(* PLC project Untitled1, Beckhoff Automation GmbH TwinCAT PLC Control 3.5.13.21 *)
(* stored: creationDateTime 2022-05-06T13:52:37.3912797, modificationDateTime 2022-05-06T13:52:37.3942797 *)

PROGRAM AutoImported
  VAR
    Step : INT;
    StepReadEtherCATDiagnostics : INT;
    TonReadDiagnostics : TON;
    sError : STRING;
    FB_EcCoESdoWrite1 : FB_EcCoESdoWrite;
    CoEWriteBuffer : DWORD;
    fbEcGetAllSlaveAbnormalStateChanges : FB_EcGetAllSlaveAbnormalStateChanges;
    fbGetAllSlaveStates : FB_EcGetAllSlaveStates;
    fbEcGetConfSlaves : FB_EcGetConfSlaves;
    fbEcGetAllSlaveCrcErrors : FB_EcGetAllSlaveCrcErrors;
    stSlaveStates : ARRAY[0..dwMaxSlaves] OF ST_EcSlaveState;
    stArrEcConfSlaveInfo : ARRAY[0..dwMaxSlaves] OF ST_EcSlaveConfigData;
    dwArrSlaveCrcCount : ARRAY[0..dwMaxSlaves] OF DWORD;
    dwArrSlaveChangeCount : ARRAY[0..dwMaxSlaves] OF DWORD;
    bExecuteFB_GetAdaptersInfo : BOOL := TRUE;  (* /////// Set IP address////////////// *)
    NICCount : INT := 2;
    NicIndex : INT := 1;
    FB_GetAdaptersInfo : FB_GetAdaptersInfo;
    fbDiagRegister : FB_IPCDiag_Register := (sNetId := '');
    fbWriteNicInfo : FB_IPCDiag_WriteParameter;
    iPrevState : INT;
    iState : INT;
    _usiModuleIndex : USINT;
    _sIPAddress : STRING;
    _sIPSubNetMask : STRING;
    _sIPGateway : STRING;
    _xDHCP : BOOL;
    rtExecuteTrig : R_TRIG;
    xBusy : BOOL;
    xError : BOOL;
    hrErrorCode : HRESULT;
    xExecute : BOOL;
    usiModuleIndex : USINT;
    sIPAddress : STRING;
    sIPSubnetMask : STRING;
    sIPGateway : STRING;
    xDHCP : BOOL;
    sCurrentNicName : STRING;
  END_VAR
  VAR CONSTANT
    dwMaxSlaves : DWORD := 50;
  END_VAR

            EtherCAT_Diagnostics();

SetIpAddress();

CASE Step OF
	0:
		//Not implimented yet.
	
	100:
		IF GVL_AutoGenerated.EtherCAT_CoEWriteExecute THEN
			Step:=Step+10;
		END_IF

		
	110:
	FB_EcCoESdoWrite1(
		sNetId:= , 
		nSlaveAddr:= , 
		nSubIndex:= , 
		nIndex:= , 
		pSrcBuf:= , 
		cbBufLen:= , 
		bExecute:= , 
		tTimeout:= , 
		bBusy=> , 
		bError=> , 
		nErrId=> );
		
	120:
		GVL_AutoGenerated.EtherCAT_CoEWriteDone:=TRUE;
END_CASE


          

METHOD EtherCAT_Diagnostics : BOOL
                  
CASE StepReadEtherCATDiagnostics OF
0:
	fbEcGetAllSlaveAbnormalStateChanges.bExecute:=FALSE;
	fbGetAllSlaveStates.bExecute:=FALSE;
	fbEcGetConfSlaves.bExecute:=FALSE;
	//fbEcGetAllSlaveCrcErrors.bError:=FALSE;
	TonReadDiagnostics(IN:=TRUE, PT:=T#1S);
	IF TonReadDiagnostics.q THEN
		TonReadDiagnostics(IN:=FALSE);
		StepReadEtherCATDiagnostics:=StepReadEtherCATDiagnostics+10;
		fbEcGetAllSlaveAbnormalStateChanges.bExecute:=TRUE;
		fbGetAllSlaveStates.bExecute:=TRUE;
		fbEcGetConfSlaves.bExecute:=TRUE;
		//fbEcGetAllSlaveCrcErrors.bError:=TRUE;
	END_IF

10:
	IF NOT fbEcGetAllSlaveAbnormalStateChanges.bBusy THEN
		StepReadEtherCATDiagnostics:=StepReadEtherCATDiagnostics+10;
		IF NOT fbEcGetAllSlaveAbnormalStateChanges.bError THEN		
			;
		ELSE
			sError:='fbEcGetAllSlaveAbnormalStateChanges';
		END_IF
	END_IF
	
20:
	IF NOT fbGetAllSlaveStates.bBusy THEN
		StepReadEtherCATDiagnostics:=StepReadEtherCATDiagnostics+10;
		IF fbGetAllSlaveStates.bError THEN
			sError:='fbGetAllSlaveStates';
		END_IF
	END_IF
	
30:
	IF NOT fbEcGetConfSlaves.bBusy THEN
		StepReadEtherCATDiagnostics:=StepReadEtherCATDiagnostics+10;
		IF fbEcGetConfSlaves.bError THEN
			sError:='fbEcGetConfSlaves';
		END_IF
	END_IF
	
40:
	IF NOT fbEcGetAllSlaveCrcErrors.bBusy THEN
		StepReadEtherCATDiagnostics:=StepReadEtherCATDiagnostics+10;
		IF fbEcGetAllSlaveCrcErrors.bError THEN			
			sError:='fbEcGetAllSlaveCrcErrors';
		END_IF
	END_IF
	
50:	//Use this step to copy all the values to PDO to be sent to the EIP network
	StepReadEtherCATDiagnostics:=0;
	GVL_AutoGenerated.EtherCATChangeCount[1]:=DWORD_TO_UINT(dwArrSlaveChangeCount[1]);
END_CASE


FB_EcCoESdoWrite1(
	sNetId:= F_CreateAmsNetId(nIds := GVL_AutoGenerated.EtherCAT_NetId) , 
	nSlaveAddr:=GVL_AutoGenerated.EtherCAT_CoEWriteSlaveAddr , 
	nSubIndex:=GVL_AutoGenerated.EtherCAT_CoEWriteSubIndex , 
	nIndex:= GVL_AutoGenerated.EtherCAT_CoEWriteIndex, 
	pSrcBuf:=ADR(CoEWriteBuffer) , 
	cbBufLen:=SIZEOF(CoEWriteBuffer) , 
	bBusy=> , 
	bError=>GVL_AutoGenerated.EtherCAT_CoEWriteError , 
	nErrId=> );

	
fbEcGetAllSlaveAbnormalStateChanges(
	sNetId:= F_CreateAmsNetId(nIds := GVL_AutoGenerated.EtherCAT_NetId), 
	pAddrBuf:= ADR(dwArrSlaveChangeCount), 
	cbBufLen:= SIZEOF(dwArrSlaveChangeCount), 
	bExecute:= , 
	tTimeout:= , 
	bBusy=> , 
	bError=> , 
	nErrId=> , 
	nSlaves=> );

fbGetAllSlaveStates(
	sNetId		:=  F_CreateAmsNetId(nIds := GVL_AutoGenerated.EtherCAT_NetId),
	pStateBuf	:= ADR(stSlaveStates),
	cbBufLen	:= SIZEOF(stSlaveStates),
	//bExecute	:=TRUE ,
	tTimeout	:= T#2s);

fbEcGetConfSlaves(bExecute:=FALSE);
fbEcGetConfSlaves(
	sNetId:=F_CreateAmsNetId(nIds := GVL_AutoGenerated.EtherCAT_NetId),
	pArrEcConfSlaveInfo:=ADR(stArrEcConfSlaveInfo) ,
	cbBufLen:=SIZEOF(stArrEcConfSlaveInfo) ,
	//bExecute:=TRUE ,
	tTimeout:=T#2s  );

fbEcGetAllSlaveCrcErrors(bExecute:=FALSE);
fbEcGetAllSlaveCrcErrors(
	sNetId:=F_CreateAmsNetId(nIds := GVL_AutoGenerated.EtherCAT_NetId) ,
	pCrcErrorBuf:=ADR(dwArrSlaveCrcCount) ,
	cbBufLen:=SIZEOF(dwArrSlaveCrcCount) ,
	//bExecute:=TRUE 
);
	
                
END_METHOD

METHOD SetIpAddress : BOOL
                  rtExecuteTrig(clk:= xExecute);
usiModuleIndex;
//sIPAddress:=GVL_Constants_AutoGenerated.PLCIPAddress;
//sIPSubnetMask:='255.255.255.0';
//xDHCP:=false;
//sIPAddress := PLCIPAddress001;

FB_GetAdaptersInfo.arrAdapters[0].bDhcpEnabled;
FB_GetAdaptersInfo.arrAdapters[1].bDhcpEnabled;
FB_GetAdaptersInfo.arrAdapters[0].sIpAddr;
FB_GetAdaptersInfo.arrAdapters[1].sIpAddr;
FB_GetAdaptersInfo.arrAdapters[1].physAddr;



FB_GetAdaptersInfo(
	sNetID:= , 
	bExecute:=bExecuteFB_GetAdaptersInfo , 
	tTimeout:= , 
	bBusy=> , 
	bError=> , 
	nErrID=> , 
	arrAdapters=> , 
	nCount=> , 
	nGet=> );

CASE iState OF
	0:	// Init
		IF NOT fbDiagRegister.bBusy THEN
			fbDiagRegister(bExecute:=TRUE); // need to be executed once
		ELSE
			fbDiagRegister(bExecute:=FALSE);
		END_IF
		IF NOT fbDiagRegister.bBusy AND NOT FB_GetAdaptersInfo.bBusy THEN
			iPrevState:= iState;
			iState := SEL(fbDiagRegister.bError, 1, 99);
			bExecuteFB_GetAdaptersInfo:=FALSE;
		END_IF
		
	1:	// Wait for execute
		IF NicIndex <= NICCount THEN
			iPrevState:= iState;
			iState:= iState+1;
			usiModuleIndex := INT_TO_USINT(NicIndex);
			sCurrentNicName := FB_GetAdaptersInfo.arrAdapters[NicIndex-1].sDescription;
			IF sCurrentNicName = 'X001' THEN		
				//usiModuleIndex:=1;
				IF PLCIPAddress001 = 'DHCP' THEN
					xDHCP:=TRUE;
				ELSE
					sIPSubnetMask:='255.255.255.0';
					xDHCP:=FALSE;
					sIPAddress := PLCIPAddress001;
				END_IF
			END_IF
			IF sCurrentNicName = 'X000' THEN
				//usiModuleIndex:=0;
				IF PLCIPAddress000 = 'DHCP' THEN
					xDHCP:=TRUE;
				ELSE
					sIPSubnetMask:='255.255.255.0';
					xDHCP:=FALSE;
					sIPAddress := PLCIPAddress000;
				END_IF		
			END_IF
		END_IF
	
	2:
	
		fbWriteNicInfo(bExecute:= FALSE, fbRegister:= fbDiagRegister);
		hrErrorCode:= 0;
		xBusy:= TRUE;
		xError:= FALSE;
		IF usiModuleIndex > 0 
			AND (xDHCP OR (sIPAddress <> '' AND sIPSubnetMask <> '')) THEN
				_usiModuleIndex:= usiModuleIndex;
				_sIPAddress:= sIPAddress;
				_sIPSubNetMask:= sIPSubnetMask;
				_sIPGateway:= sIPGateway;
				_xDHCP:= xDHCP;
				iPrevState:= iState;
				iState:= 20;					
		ELSE
			iPrevState:= iState;
			iState:= 99;	
		END_IF				


		
	20:	// Write DHCP
		fbWriteNicInfo(
			bExecute:= TRUE, 
			eParameterKey:= E_IPCDiag_ParameterKey.NIC_DHCP, 
			pBuffer:= ADR(_xDHCP), 
			nBufferSize:= SIZEOF(_xDHCP), 
			nModuleIdx:= _usiModuleIndex, 
			nListIdx:= , 
			tTimeout:= T#5S, 
			sNetId:= '', 
			xReserved:= , 
			fbRegister:= fbDiagRegister, 
			bBusy=> , 
			bError=> , 
			hrErrorCode=> , 
			ipErrorMessage=> );
	
		IF NOT fbWriteNicInfo.bBusy THEN
			IF NOT fbWriteNicInfo.bError THEN
				fbWriteNicInfo(bExecute:= FALSE, fbRegister:= fbDiagRegister);
				iPrevState:= iState;
				iState:= iState + 10;
				IF _xDHCP THEN
					iState:= 60;
				END_IF
			ELSE
				iPrevState:= iState;
				iState:= 99;
			END_IF
		END_IF
		
	30: // Write IP Address
		fbWriteNicInfo(
			bExecute:= TRUE, 
			eParameterKey:= E_IPCDiag_ParameterKey.NIC_IPv4Address, 
			pBuffer:= ADR(_sIPAddress), 
			nBufferSize:= SIZEOF(_sIPAddress), 
			nModuleIdx:= _usiModuleIndex, 
			nListIdx:= , 
			tTimeout:= T#5S, 
			sNetId:= '', 
			xReserved:= , 
			fbRegister:= fbDiagRegister, 
			bBusy=> , 
			bError=> , 
			hrErrorCode=> , 
			ipErrorMessage=> );
	
		IF NOT fbWriteNicInfo.bBusy THEN
			IF NOT fbWriteNicInfo.bError THEN
				fbWriteNicInfo(bExecute:= FALSE, fbRegister:= fbDiagRegister);
				iPrevState:= iState;
				iState:= iState + 10;
			ELSE
				iPrevState:= iState;
				iState:= 99;
			END_IF
		END_IF	
	
	40:	// Write Subnet Mask
		fbWriteNicInfo(
			bExecute:= TRUE, 
			eParameterKey:= E_IPCDiag_ParameterKey.NIC_IPv4SubnetMask, 
			pBuffer:= ADR(_sIPSubNetMask), 
			nBufferSize:= SIZEOF(_sIPSubNetMask), 
			nModuleIdx:= _usiModuleIndex, 
			nListIdx:= , 
			tTimeout:= T#5S, 
			sNetId:= '', 
			xReserved:= , 
			fbRegister:= fbDiagRegister, 
			bBusy=> , 
			bError=> , 
			hrErrorCode=> , 
			ipErrorMessage=> );
	
		IF NOT fbWriteNicInfo.bBusy THEN
			IF NOT fbWriteNicInfo.bError THEN
				fbWriteNicInfo(bExecute:= FALSE, fbRegister:= fbDiagRegister);
				iPrevState:= iState;
				iState:= iState + 10;
			ELSE
				iPrevState:= iState;
				iState:= 99;
			END_IF
		END_IF		
	
	50:	// Write Gateway
		fbWriteNicInfo(
			bExecute:= TRUE, 
			eParameterKey:= E_IPCDiag_ParameterKey.NIC_IPv4DefGateway, 
			pBuffer:= ADR(_sIPGateway), 
			nBufferSize:= SIZEOF(_sIPGateway), 
			nModuleIdx:= _usiModuleIndex, 
			nListIdx:= , 
			tTimeout:= T#5S, 
			sNetId:= '', 
			xReserved:= , 
			fbRegister:= fbDiagRegister, 
			bBusy=> , 
			bError=> , 
			hrErrorCode=> , 
			ipErrorMessage=> );
	
		IF NOT fbWriteNicInfo.bBusy THEN
			IF NOT fbWriteNicInfo.bError THEN
				fbWriteNicInfo(bExecute:= FALSE, fbRegister:= fbDiagRegister);
				iPrevState:= iState;
				iState:= iState + 10;
			ELSE
				iPrevState:= iState;
				iState:= 99;
			END_IF
		END_IF		
		
	60:
		xBusy:= FALSE;
		xError:= FALSE;
		iPrevState:= iState;
		iState:= 0;
		NicIndex:=NicIndex+1;
		bExecuteFB_GetAdaptersInfo:=TRUE;
	
	99:
		xBusy:= FALSE;
		xError:= TRUE;
		hrErrorCode:= fbWriteNicInfo.hrErrorCode;
		IF NOT xExecute THEN
			iPrevState:= iState;
			iState:= 0;
		END_IF
	
END_CASE

                
END_METHOD
END_PROGRAM
